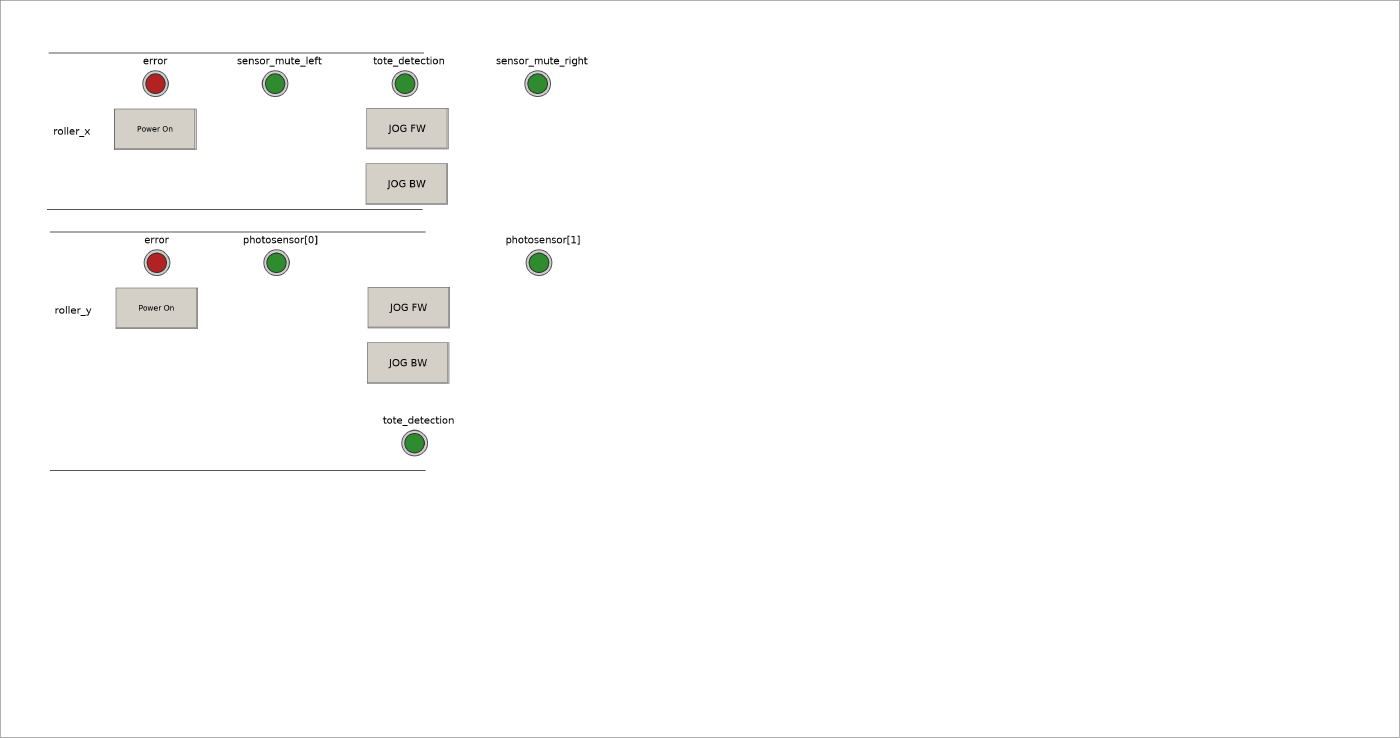
VISUALIZATION v_io_loading  // 2048x1080
    Lamp1 (570,100 45x45), variable: GVL.fb_loading.photo_sensor_tote_detection, style: Lamp-Lamp1-Green
    Label (526,76 145x26), "tote_detection"
    Lamp1 (205,100 45x45), variable: GVL.fb_loading.roller_x.roller.err, style: Lamp-Lamp1-Red
    Label (161,76 132x26), "error"
    Line (71,77) (620,77)
    Button (536,158 120x60), "JOG FW", colour toggle: GVL.fb_loading.roller_x.roller.forward
        OnMouseDown: execute { GVL.fb_loading.roller_x.roller.forward	:= TRUE; }
        OnMouseUp: execute { GVL.fb_loading.roller_x.roller.forward	:= FALSE; }
    Button (535,239 120x60), "JOG BW", colour toggle: GVL.fb_loading.roller_x.roller.backward
        OnMouseDown: execute { GVL.fb_loading.roller_x.roller.backward	:= TRUE; }
        OnMouseUp: execute { GVL.fb_loading.roller_x.roller.backward	:= FALSE; }
    Button (167,159 120x60), "Power On", colour toggle: GVL.fb_loading.roller_x.roller.Power
        toggle GVL.fb_loading.roller_x.roller.Power
    Line (69,306) (618,306)
    Lamp1 (380,100 45x45), variable: GVL.fb_loading.roller_x.photo_sensor_mute_left, style: Lamp-Lamp1-Green
    Label (336,76 145x26), "sensor_mute_left"
    Lamp1 (764,100 45x45), variable: GVL.fb_loading.roller_x.photo_sensor_mute_right, style: Lamp-Lamp1-Green
    Label (720,76 145x26), "sensor_mute_right"
    Label (39,179 132x26), "roller_x"
    Lamp1 (584,626 45x45), variable: GVL.fb_loading.roller_y.roller.sensor, style: Lamp-Lamp1-Green
    Label (540,602 145x26), "tote_detection"
    Lamp1 (207,362 45x45), variable: GVL.fb_loading.roller_y.roller.err, style: Lamp-Lamp1-Red
    Label (163,338 132x26), "error"
    Line (73,339) (622,339)
    Button (538,420 120x60), "JOG FW", colour toggle: GVL.fb_loading.roller_y.roller.forward
        OnMouseDown: execute { GVL.fb_loading.roller_y.roller.forward	:= TRUE; }
        OnMouseUp: execute { GVL.fb_loading.roller_y.roller.forward	:= FALSE; }
    Button (537,501 120x60), "JOG BW", colour toggle: GVL.fb_loading.roller_y.roller.backward
        OnMouseDown: execute { GVL.fb_loading.roller_y.roller.backward	:= TRUE; }
        OnMouseUp: execute { GVL.fb_loading.roller_y.roller.backward	:= FALSE; }
    Button (169,421 120x60), "Power On", colour toggle: GVL.fb_loading.roller_y.roller.Power
        toggle GVL.fb_loading.roller_y.roller.Power
    Line (73,688) (622,688)
    Lamp1 (382,362 45x45), variable: GVL.fb_loading.roller_y.photo_sensor[0], style: Lamp-Lamp1-Green
    Label (338,338 145x26), "photosensor[0]"
    Lamp1 (766,362 45x45), variable: GVL.fb_loading.roller_y.photo_sensor[1], style: Lamp-Lamp1-Green
    Label (722,338 145x26), "photosensor[1]"
    Label (41,441 132x26), "roller_y"
END_VISUALIZATION

(* stored: Version 1.1.0.1, ProductVersion 3.1.4024.12
   Visu v_io_loading: Id {cd18c918-ee0d-4af8-834e-d168810db6db} *)
